TYPE ST_AteqF6_Device :
STRUCT
	stIn  : ST_AteqF6_Read;
    stOut : ST_AteqF6_Write;
END_STRUCT
END_TYPE

(* stored: Version 1.1.0.1, ProductVersion 3.1.4024.15
   DUT ST_AteqF6_Device: Id {7ce7ac0c-1c92-4cec-a3bd-bf1f5c9de48e} *)
